# EPICS autosave request: iocBoot/iocrsfsl/auto_settings_RSFSV.req
file "RSFSV_settings.req",                P=$(P),  R=$(R)
